FUNCTION_BLOCK FB_Ventilation
VAR_INPUT
END_VAR
VAR_OUTPUT
END_VAR
VAR
END_VAR

END_FUNCTION_BLOCK

(* stored: Version 1.1.0.1, ProductVersion 3.1.4024.10
   POU FB_Ventilation: Id {94cdc637-68fc-4965-95c2-bd12607af2ac}, SpecialFunc None *)
